# EPICS autosave request: iocBoot/ioc13Galil_test/Galil_settings.req
file "CARS_8_motor_settings.req",      P=$(P)
file "pseudoMotor_settings.req",        P=$(P), M=pm1
file "pseudoMotor_settings.req",        P=$(P), M=pm2
file "pseudoMotor_settings.req",        P=$(P), M=pm3
file "pseudoMotor_settings.req",        P=$(P), M=pm4

file "galil_motor_extras.req",          P=$(P)Galil1:, M=m1
file "galil_motor_extras.req",          P=$(P)Galil1:, M=m2
file "galil_motor_extras.req",          P=$(P)Galil1:, M=m3
file "galil_motor_extras.req",          P=$(P)Galil1:, M=m4
file "galil_motor_extras.req",          P=$(P)Galil1:, M=m5
file "galil_motor_extras.req",          P=$(P)Galil1:, M=m6
file "galil_motor_extras.req",          P=$(P)Galil1:, M=m7
file "galil_motor_extras.req",          P=$(P)Galil1:, M=m8
